CONFIGURATION Device
  RESOURCE Application ON PLC
    VAR_GLOBAL  (* GVL - ============================================================================== GVL: 全局变量表（核心数据枢纽） 作用: - 三轴 CANopen 过程映像（%QX/%IX/%QD/%ID 与驱动器 PDO 交换） - 本控/远控轴命令结构 Axis1/2/3 Local & Remote - 时统、跟踪接收机、故障与显示相关全局量 轴对应: Axis1=俯仰El Axis2=方位Az Axis3=倾斜Ti 主要读写: *_ctrl_1, *_Ctrl_FB, SecurityCheck, Modbus_Slave, READ_485 复制到 CODESYS: 仅粘贴 VAR_GLOBAL ... END_VAR，保留所有 AT 地址不变 ============================================================================== *)
      bElCtrlBit0 AT %QX4.0 : BOOL;  (* 控制字位0，上电序列用 *)
      bElCtrlBit1 AT %QX4.1 : BOOL;  (* 控制字位1 *)
      bElCtrlBit2 AT %QX4.2 : BOOL;  (* 控制字位2 *)
      bElCtrlBit3 AT %QX4.3 : BOOL;  (* 控制字位3，下电时清 *)
      bElCtrlBit4 AT %QX4.4 : BOOL;  (* 控制字位4 *)
      bElCtrlBit5 AT %QX4.5 : BOOL;  (* 控制字位5 *)
      bElCtrlBit7 AT %QX4.7 : BOOL;  (* 控制字位7，故障复位脉冲用 *)
      bElCtrlBit8 AT %QX5.0 : BOOL;  (* 快速停止/减速停止请求 *)
      diElTargetVel AT %QD2 : DINT;  (* 目标速度 raw（524288/圈） *)
      diElTargetPos AT %QD3 : DINT;  (* 目标位置 raw *)
      diElTargetAcc AT %QD4 : UDINT;  (* 加速度 raw *)
      diElTargetDec AT %QD5 : UDINT;  (* 减速度 raw *)
      bElStsBit0 AT %IX4.0 : BOOL;  (* 状态字位0，参与“已使能”判断 *)
      bElStsBit1 AT %IX4.1 : BOOL;  (* 状态字位1 *)
      bElStsBit2 AT %IX4.2 : BOOL;  (* 状态字位2 *)
      bElStsBit3 AT %IX4.3 : BOOL;  (* 状态字位3，故障位→Axis1Status.Error *)
      bElStsBit10 AT %IX5.2 : BOOL;  (* 状态字扩展位 *)
      bElStsBit12 AT %IX5.4 : BOOL;  (* 状态字扩展位 *)
      diElActVel AT %ID2 : DINT;  (* 实际速度 raw → rFctVelReal_1 *)
      diElActPos AT %ID3 : DINT;  (* 实际位置 raw → rFctPosReal_1 *)
      siElMode AT %QB6 : UINT;  (* 驱动器模式字写入 *)
      eElErrorcode AT %IW3 : UINT;  (* 驱动器故障码，如 16#8130 心跳 *)
      bAzCtrlBit0 AT %QX24.0 : BOOL;  (* ----- 方位轴 Az：CANopen 输出 %QX24/%QD7-10 ----- *)
      bAzCtrlBit1 AT %QX24.1 : BOOL;
      bAzCtrlBit2 AT %QX24.2 : BOOL;
      bAzCtrlBit3 AT %QX24.3 : BOOL;
      bAzCtrlBit4 AT %QX24.4 : BOOL;
      bAzCtrlBit5 AT %QX24.5 : BOOL;
      bAzCtrlBit7 AT %QX24.7 : BOOL;
      bAzCtrlBit8 AT %QX25.0 : BOOL;
      diAzTargetVel AT %QD7 : DINT;
      diAzTargetPos AT %QD8 : DINT;
      diAzTargetAcc AT %QD9 : UDINT;
      diAzTargetDec AT %QD10 : UDINT;
      bAzStsBit0 AT %IX24.0 : BOOL;  (* ----- 方位轴 Az：CANopen 输入 %IX24/%ID7-8 ----- *)
      bAzStsBit1 AT %IX24.1 : BOOL;
      bAzStsBit2 AT %IX24.2 : BOOL;
      bAzStsBit3 AT %IX24.3 : BOOL;
      bAzStsBit10 AT %IX25.2 : BOOL;
      bAzStsBit12 AT %IX25.4 : BOOL;
      diAzActVel AT %ID7 : DINT;
      diAzActPos AT %ID8 : DINT;
      siAzMode AT %QB26 : UINT;
      eAzErrorcode AT %IW13 : UINT;
      bTiCtrlBit0 AT %QX44.0 : BOOL;  (* ----- 倾斜轴 Ti：CANopen 输出 %QX44/%QD12-15 ----- *)
      bTiCtrlBit1 AT %QX44.1 : BOOL;
      bTiCtrlBit2 AT %QX44.2 : BOOL;
      bTiCtrlBit3 AT %QX44.3 : BOOL;
      bTiCtrlBit4 AT %QX44.4 : BOOL;
      bTiCtrlBit5 AT %QX44.5 : BOOL;
      bTiCtrlBit7 AT %QX44.7 : BOOL;
      bTiCtrlBit8 AT %QX45.0 : BOOL;
      diTiTargetVel AT %QD12 : DINT;
      diTiTargetPos AT %QD13 : DINT;
      diTiTargetAcc AT %QD14 : UDINT;
      diTiTargetDec AT %QD15 : UDINT;
      bTiStsBit0 AT %IX44.0 : BOOL;  (* ----- 倾斜轴 Ti：CANopen 输入 %IX44/%ID12-13 ----- *)
      bTiStsBit1 AT %IX44.1 : BOOL;
      bTiStsBit2 AT %IX44.2 : BOOL;
      bTiStsBit3 AT %IX44.3 : BOOL;
      bTiStsBit10 AT %IX45.2 : BOOL;
      bTiStsBit12 AT %IX45.4 : BOOL;
      diTiActVel AT %ID12 : DINT;
      diTiActPos AT %ID13 : DINT;
      siTiMode AT %QB46 : UINT;
      eTiErrorcode AT %IW23 : UINT;
      dDelTime : DINT;  (* GNSS 与本地时钟偏差 (ms)，TimeCase 校正 *)
      stGNSS_Timestap : ULINT;  (* GNSS 时间戳 (ms)，GPRMC_1 写入 *)
      dRealTime : ULINT;  (* 当前应用时间 (ms)，RealTimePosCal 生成 *)
      bLocalCtrl : BOOL;  (* TRUE=本控 FALSE=远控（Modbus/HMI） *)
      bError_Reset : BOOL;  (* 故障复位请求，SecurityCheck/Modbus *)
      Error_code : INT;  (* 应用层故障码，上报 Modbus IR[5] *)
      Axis1Local : AxisCrtlStruct;  (* 本控命令 *)
      Axis1Remote : AxisCrtlStruct;  (* 远控命令（SecurityCheck←Modbus） *)
      Axis1Status : AxisStatus;  (* 俯仰状态 *)
      Axis1Visible : AxisVisible;  (* 俯仰 HMI 显示 *)
      rFctPosReal_1 : LREAL;  (* 俯仰实际位置 (deg) *)
      rFctVelReal_1 : LREAL;  (* 俯仰实际速度 (deg/s) *)
      rFctAccReal_1 : LREAL;  (* 俯仰加速度（显示/备用） *)
      rFctDecReal_1 : LREAL;  (* 俯仰减速度（显示/备用） *)
      Axis2Local : AxisCrtlStruct;  (* ----- 轴2 方位 Az：逻辑控制结构 ----- *)
      Axis2Remote : AxisCrtlStruct;
      Axis2Status : AxisStatus;
      Axis2Visible : AxisVisible;
      rFctPosReal_2 : REAL;  (* 方位实际位置 (deg)，常为编码器×-1 *)
      rFctVelReal_2 : LREAL;
      rFctAccReal_2 : LREAL;
      rFctDecReal_2 : LREAL;
      Axis3Local : AxisCrtlStruct;  (* ----- 轴3 倾斜 Ti：逻辑控制结构 ----- *)
      Axis3Remote : AxisCrtlStruct;
      Axis3Status : AxisStatus;
      Axis3Visible : AxisVisible;
      rFctPosReal_3 : REAL;
      rFctVelReal_3 : LREAL;
      rFctAccReal_3 : LREAL;
      rFctDecReal_3 : LREAL;
      bStartTrack : BOOL;  (* 自跟踪总使能，SecurityCheck 根据 ACU 处理 *)
      Chan1AGC : REAL;  (* 通道1 自动增益 (dB 等) *)
      Chan1Ua : REAL;  (* 通道1 方位误差电压 *)
      Chan1Ue : REAL;  (* 通道1 俯仰误差电压 *)
      Chan1Lock : BOOL;  (* 通道1 锁定（AGC>门限） *)
      Chan1Online : BOOL;  (* 通道1 在线 *)
      Chan2AGC : REAL;  (* 通道2 AGC *)
      Chan2Ua : REAL;
      Chan2Ue : REAL;
      Chan2Lock : BOOL;
      Chan2Online : BOOL;
      Chanthreshold : REAL;  (* AGC 锁定门限，Modbus HR[43] 可写 *)
      AzV : AxisCrtlStruct;  (* ----- 可视化/备用轴结构（部分画面绑定）----- *)
      ElV : AxisCrtlStruct;
      TiV : AxisCrtlStruct;
      iTest : INT;  (* 测试用 *)
      a : INT;  (* 测试用 *)
      iVisualSwitch : INT;  (* 画面切换 *)
      bAzVisable : BOOL;  (* 方位显示使能 *)
      bElVisable : BOOL;  (* 俯仰显示使能 *)
      bTlVisable : BOOL;  (* 倾斜显示使能 *)
      bLocalAutoTrackVis : BOOL;  (* 本控自跟踪画面 *)
      bStartLocalAutoTrack : BOOL;  (* 本控启动自跟踪 *)
      bRemoteTimeLock : BOOL;  (* 远控时间锁定 *)
      Ti : REAL;  (* 倾斜显示角 *)
      El : REAL;  (* 俯仰显示角 *)
      bTimeSwich : BOOL;  (* 时间源选择：FALSE=GNSS TRUE=Modbus UTC *)
      rvAzKpBase : REAL;  (* 方位 Kp 显示/调试镜像 *)
      rvAzKiBase : REAL;
      rvAzKpscale : REAL;
      rvAzKiscale : REAL;
      rvElKpBase : REAL;
      rvElKiBase : REAL;
      rvElKpscale : REAL;
      rvElKiscale : REAL;
      rvAzKpMax : REAL;
      rvAzKiMax : REAL;
      rvElKpMax : REAL;
      rvElKiMax : REAL;
      rvAzThre : REAL;
      rvElThre : REAL;
      bTrackingModeTemp : BOOL;  (* 跟踪模式临时 *)
      rAzScanRangeTemp : REAL;  (* 扫描范围临时 *)
      rElScanRangeTemp : REAL;
      rErrorTherTemp : REAL;  (* 误差门限临时 *)
      rStepTemp : REAL;  (* 步长临时 *)
    END_VAR
    {attribute 'qualified_only'}
    {attribute 'checksumnoinit_override' := '3797087048'}
    {attribute 'init_related_code' := '4f941375-a68b-4e0d-aefe-3b3eb66ff5e0'}
    VAR_GLOBAL PERSISTENT  (* PersistentVars - ============================================================================== GVL: PersistentVars（掉电保持） 作用: 上电后仍保留的标定、PID 基准、扫描/跟踪参数 写入: 通常由 HMI、首次标定或 Modbus 相关逻辑写入 读取: vpid、SecurityCheck、自跟踪/扫描程序 ============================================================================== *)
      {attribute 'order_in_persistent_editor' := '0'}
      TiOffset : REAL;  (* 倾斜轴零点/偏置 (deg) *)
      {attribute 'order_in_persistent_editor' := '1'}
      ElOffset : REAL;  (* 俯仰轴零点/偏置 (deg) *)
      {attribute 'order_in_persistent_editor' := '2'}
      rAzKpBase : REAL;  (* 方位 vpid 基础 Kp *)
      {attribute 'order_in_persistent_editor' := '3'}
      rAzKiBase : REAL;  (* 方位 vpid 基础 Ki *)
      {attribute 'order_in_persistent_editor' := '4'}
      rAzKpscale : REAL;  (* 方位 Kp 缩放 *)
      {attribute 'order_in_persistent_editor' := '5'}
      rAzKiscale : REAL;  (* 方位 Ki 缩放 *)
      {attribute 'order_in_persistent_editor' := '6'}
      rElKpBase : REAL;  (* 俯仰 vpid 基础 Kp *)
      {attribute 'order_in_persistent_editor' := '7'}
      rElKiBase : REAL;  (* 俯仰 vpid 基础 Ki *)
      {attribute 'order_in_persistent_editor' := '8'}
      rElKpscale : REAL;  (* 俯仰 Kp 缩放 *)
      {attribute 'order_in_persistent_editor' := '9'}
      rElKiscale : REAL;  (* 俯仰 Ki 缩放 *)
      {attribute 'order_in_persistent_editor' := '10'}
      rAzKpMax : REAL;  (* 方位 Kp 上限 *)
      {attribute 'order_in_persistent_editor' := '11'}
      rAzKiMax : REAL;  (* 方位 Ki 上限 *)
      {attribute 'order_in_persistent_editor' := '12'}
      rElKpMax : REAL;  (* 俯仰 Kp 上限 *)
      {attribute 'order_in_persistent_editor' := '13'}
      rElKiMax : REAL;  (* 俯仰 Ki 上限 *)
      {attribute 'order_in_persistent_editor' := '14'}
      rAzThre : REAL;  (* 方位 vpid 速度阈值 *)
      {attribute 'order_in_persistent_editor' := '15'}
      rElThre : REAL;  (* 俯仰 vpid 速度阈值 *)
      {attribute 'order_in_persistent_editor' := '16'}
      bTrackingMode : BOOL;  (* 跟踪模式开关（保持） *)
      {attribute 'order_in_persistent_editor' := '17'}
      rAzScanRange : REAL;  (* 方位扫描范围 *)
      {attribute 'order_in_persistent_editor' := '18'}
      rElScanRange : REAL;  (* 俯仰扫描范围 *)
      {attribute 'order_in_persistent_editor' := '19'}
      bSearchType : BOOL;  (* 搜索类型选择 *)
      {attribute 'order_in_persistent_editor' := '20'}
      rErrorThre : REAL;  (* 跟踪/搜索误差门限 *)
      {attribute 'order_in_persistent_editor' := '21'}
      rStartThre : REAL;  (* 自跟踪启动 AGC 门限（SecurityCheck 等） *)
      {attribute 'order_in_persistent_editor' := '22'}
      rStep : REAL;  (* 搜索步长 (deg) *)
    END_VAR
    TASK MainTask(INTERVAL := T#50ms, PRIORITY := 10);
    TASK SerialCom(INTERVAL := T#5ms, PRIORITY := 1);
    TASK Canopen(INTERVAL := T#10ms, PRIORITY := 0);
    TASK Task(INTERVAL := T#50ms, PRIORITY := 31);
    TASK VISU_TASK(INTERVAL := T#100ms, PRIORITY := 31);
    PROGRAM Modbus_Slave WITH MainTask : Modbus_Slave;
    PROGRAM READ_485 WITH SerialCom : READ_485;
    PROGRAM GPRMC_1 WITH SerialCom : GPRMC_1;
    PROGRAM TimeAdd WITH Canopen : TimeAdd;
    PROGRAM AutoTrackingCal WITH Canopen : AutoTrackingCal;
    PROGRAM El_ctrl_1 WITH Canopen : El_ctrl_1;
    PROGRAM Az_ctrl_1 WITH Canopen : Az_ctrl_1;
    PROGRAM Ti_ctrl_1 WITH Canopen : Ti_ctrl_1;
    PROGRAM RealTimePosCal WITH Canopen : RealTimePosCal;
    PROGRAM SecurityCheck WITH Canopen : SecurityCheck;
    PROGRAM VisuElems.Visu_Prg WITH VISU_TASK : VisuElems.Visu_Prg;
  END_RESOURCE
END_CONFIGURATION

CONFIGURATION GCAN_IoDrv
END_CONFIGURATION

CONFIGURATION GCAN_IoMDP
END_CONFIGURATION

CONFIGURATION GC5016_Digital_Input_Output
END_CONFIGURATION

CONFIGURATION CANbus
END_CONFIGURATION

CONFIGURATION CANopen_Manager
END_CONFIGURATION

CONFIGURATION eDriver_El
END_CONFIGURATION

CONFIGURATION eDriver_Az
END_CONFIGURATION

CONFIGURATION eDriver_Ti
END_CONFIGURATION

CONFIGURATION SoftMotion General Axis Pool
END_CONFIGURATION
